(* Logix 5000 project; controller PBS_Perfusion vendor 1 type 14 code 217 rev 32.14; software revision 32.03; part 4 of 27 *)
(* tags used below, declared in another part *)
   ONS : DINT[3];
   REAL : DINT;

ADD_ON_INSTRUCTION AMP_Q_Segment_Execute   (* revision 1.0 *)
// Applied Motion - Q Segment Execute AOI
// Help:
// The SCL Command Execute AOI executes selected SCL commands (as listed under “Available SCL Commands” in the Host Command Reference).
VAR_IN_OUT
   Input : DINT[14]; {required}   // Drive Input Assembly
   Output : DINT[16]; {required}   // Drive Output Assembly
        [0]   // Command Word
        [1]   // Jog Speed (0.25 rev/min)
        [2]   // Jog Acceleration (10 rev/s/s)
        [3]   // Jog Deceleration (10 rev/s/s)
        [4]   // Point-to-Point Velocity (0.25 rev/min)
        [5]   // Point-to-Point Acceleration (10 rev/s/s)
        [6]   // Point-to-Point Deceleration (10 rev/s/s)
        [7]   // Point-to-Point Distance (Motor steps)
        [9]   // (2x ASCII Letters in 16 lower word)
        [10]   // Data/Register 1
        [11]   // Data/Register 2
END_VAR
VAR_INPUT
   RPI : DINT := 100; {visible}   // Drive Connection Request Packet Interval (milliseconds)
   LoadAndExec : BOOL; {required}   // Load and Execute the specified Q segment (edge triggered)
   Q_Segment : DINT; {required}   // Q Segment to Load and Execute
END_VAR
VAR_OUTPUT
   Sent : BOOL; {access Read Only, visible}   // Command has been sent to drive
   In_Progress : BOOL; {access Read Only, visible}   // In progress = sending command
   Done : BOOL; {access Read Only, visible}   // Command sent
   Error : BOOL; {access Read Only, visible}   // Command failed to be sent
   State : DINT := 10; {access Read Only}   // Internal state of progress
END_VAR
VAR
   Loc_StatusCode : AMP_Status_Word;
   Loc_CommandOff_Timer : TIMER;   // Timer to make sure command value was 0 before sending a new command
   Loc_CommandOn_Timer : TIMER;   // Timer to make sure command value is set long enough to be sent to drive
   Loc_Input_Assembly : AMP_Input_Assembly_v2; {access None}
   Loc_Start_ONS : BOOL; {access None}
END_VAR

ROUTINE Logic   (* ladder *)
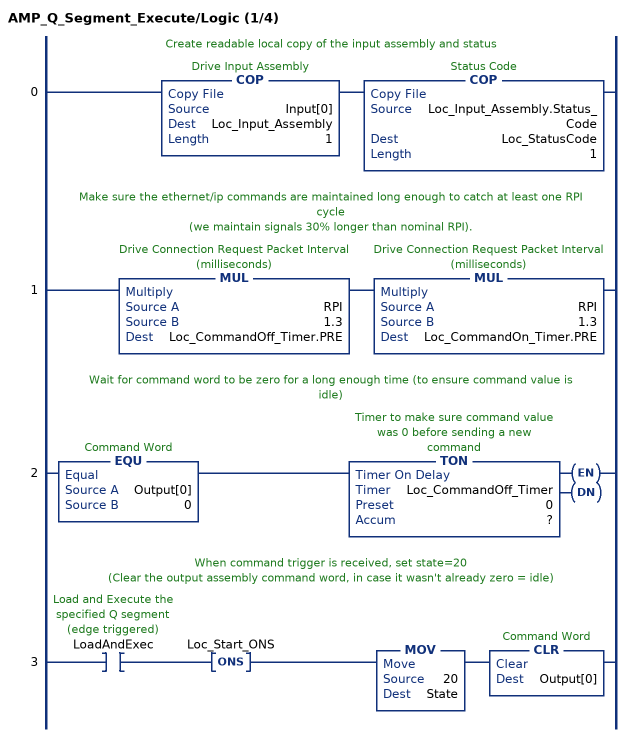
   // Create readable local copy of the input assembly and status
   0: COP(Input[0],Loc_Input_Assembly,1)COP(Loc_Input_Assembly.Status_Code,Loc_StatusCode,1);
   // Make sure the ethernet/ip commands are maintained long enough to catch at least one RPI cycle
   // (we maintain signals 30% longer than nominal RPI).
   1: MUL(RPI,1.3,Loc_CommandOff_Timer.PRE)MUL(RPI,1.3,Loc_CommandOn_Timer.PRE);
   // Wait for command word to be zero for a long enough time (to ensure command value is idle)
   2: EQU(Output[0],0)TON(Loc_CommandOff_Timer,?,?);
   // When command trigger is received, set state=20
   // (Clear the output assembly command word, in case it wasn't already zero = idle)
   3: XIC(LoadAndExec)ONS(Loc_Start_ONS)MOV(20,State)CLR(Output[0]);
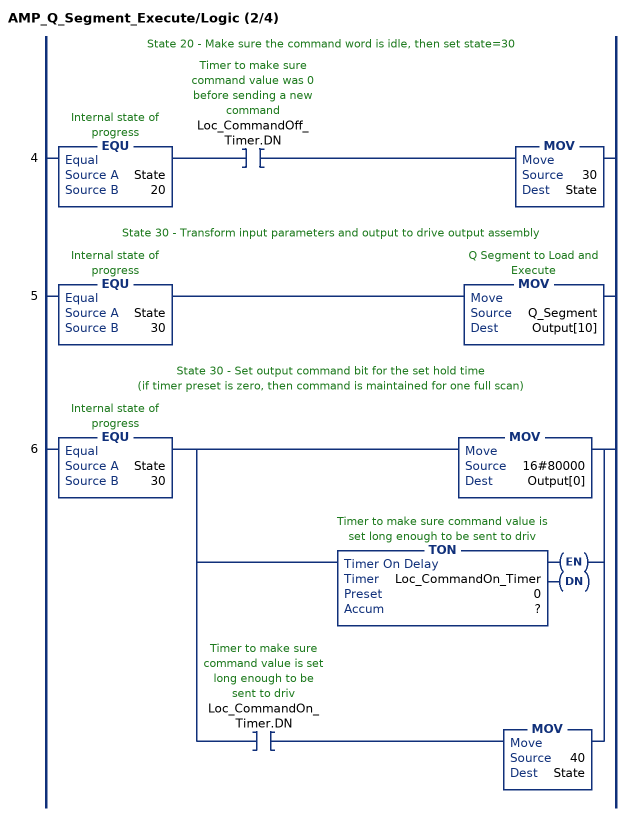
   // State 20 - Make sure the command word is idle, then set state=30
   4: EQU(State,20)XIC(Loc_CommandOff_Timer.DN)MOV(30,State);
   // State 30 - Transform input parameters and output to drive output assembly
   5: EQU(State,30)MOV(Q_Segment,Output[10]);
   // State 30 - Set output command bit for the set hold time
   // (if timer preset is zero, then command is maintained for one full scan)
   6: EQU(State,30)[MOV(16#80000,Output[0]) ,TON(Loc_CommandOn_Timer,?,?) ,XIC(Loc_CommandOn_Timer.DN) MOV(40,State) ];
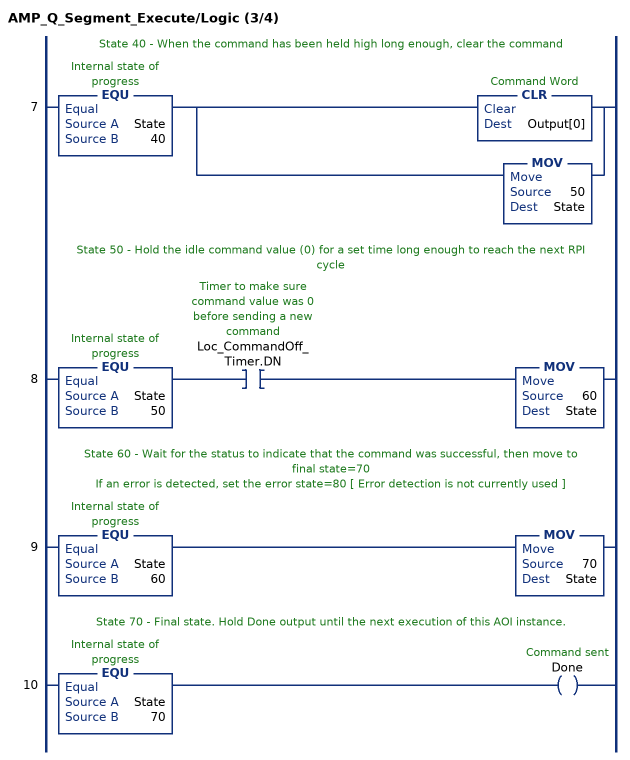
   // State 40 - When the command has been held high long enough, clear the command
   7: EQU(State,40)[CLR(Output[0]) ,MOV(50,State) ];
   // State 50 - Hold the idle command value (0) for a set time long enough to reach the next RPI cycle
   8: EQU(State,50)XIC(Loc_CommandOff_Timer.DN)MOV(60,State);
   // State 60 - Wait for the status to indicate that the command was successful, then move to final state=70
   // If an error is detected, set the error state=80 [ Error detection is not currently used ]
   9: EQU(State,60)MOV(70,State);
   // State 70 - Final state. Hold Done output until the next execution of this AOI instance.
   10: EQU(State,70)OTE(Done);
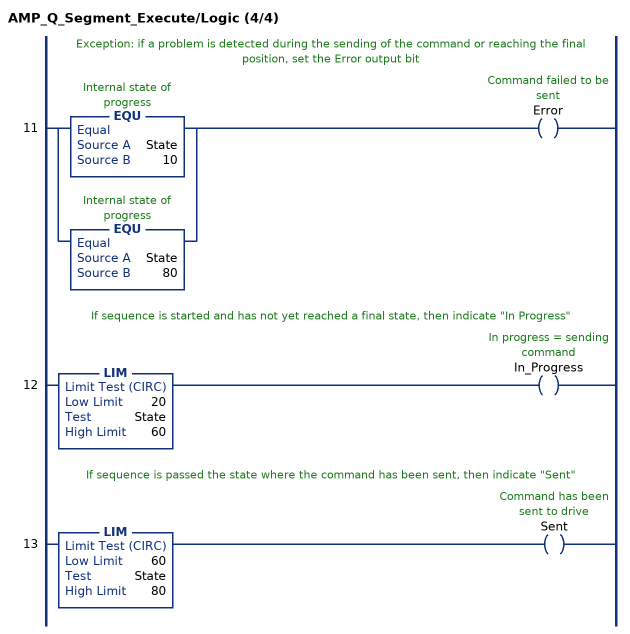
   // Exception: if a problem is detected during the sending of the command or reaching the final position, set the Error output bit
   11: [EQU(State,10) ,EQU(State,80) ]OTE(Error);
   // If sequence is started and has not yet reached a final state, then indicate "In Progress"
   12: LIM(20,State,60)OTE(In_Progress);
   // If sequence is passed the state where the command has been sent, then indicate "Sent"
   13: LIM(60,State,80)OTE(Sent);
END_ROUTINE
END_ADD_ON_INSTRUCTION

ADD_ON_INSTRUCTION AMP_Relative_Move   (* revision 1.0 *)
// Applied Motion - Relative Move AOI
// Help:
// The Relative Move AOI is used to move an axis by a specified distance (positive or negative) relative to its currently commanded position.
VAR_IN_OUT
   Input : DINT[14]; {required}   // Drive Input Assembly
   Output : DINT[16]; {required}   // Drive Output Assembly
        [0]   // Command Word
        [1]   // Jog Speed (0.25 rev/min)
        [2]   // Jog Acceleration (10 rev/s/s)
        [3]   // Jog Deceleration (10 rev/s/s)
        [4]   // Point-to-Point Velocity (0.25 rev/min)
        [5]   // Point-to-Point Acceleration (10 rev/min/s)
        [6]   // Point-to-Point Deceleration (10 rev/min/s)
        [7]   // Point-to-Point Distance (Motor steps)
        [9]   // (2x ASCII Letters in 16 lower word)
        [10]   // Data/Register 1
        [11]   // Data/Register 2
END_VAR
VAR_INPUT
   RPI : DINT := 100; {visible}   // Drive Connection Request Packet Interval (milliseconds)
   Start : BOOL; {required}   // Start the Relative Move
   Distance : DINT; {required}   // Relative Distance to Move (steps, negative = reverse)
   Speed : REAL; {required}   // Velocity of Move (rev/min)
   Acc : REAL; {required}   // Acceleration of Move (rev/s/s)
   Dec : REAL; {required}   // Deceleration (rev/s/s)
END_VAR
VAR_OUTPUT
   Sent : BOOL; {access Read Only, visible}   // Move has been sent to drive
   In_Progress : BOOL; {access Read Only, visible}   // Move in progress
   Done : BOOL; {access Read Only, visible}   // Move completed without errors - desired position reached
   Error : BOOL; {access Read Only, visible}   // Move failed to complete - drive not ready or faulted
   State : DINT := 10; {access Read Only}   // Internal state of progress
END_VAR
VAR
   Loc_StatusCode : AMP_Status_Word;
   Loc_CommandOff_Timer : TIMER;   // Timer to make sure command value was 0 before sending a new command
   Loc_CommandOn_Timer : TIMER;   // Timer to make sure command value is set long enough to be sent to drive
   Loc_Input_Assembly : AMP_Input_Assembly_v2; {access None}
   Loc_Start_ONS : BOOL; {access None}
   Loc_AlarmCode : AMP_Alarm_Word; {access None}
END_VAR

ROUTINE Logic   (* ladder *)
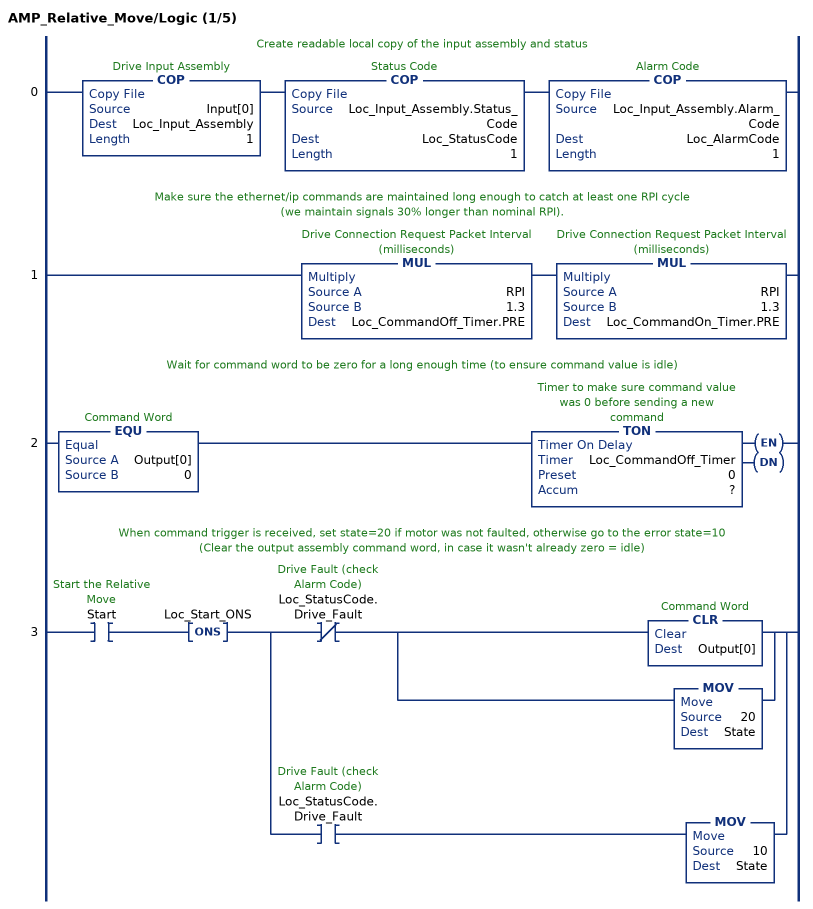
   // Create readable local copy of the input assembly and status
   0: COP(Input[0],Loc_Input_Assembly,1)COP(Loc_Input_Assembly.Status_Code,Loc_StatusCode,1)COP(Loc_Input_Assembly.Alarm_Code,Loc_AlarmCode,1);
   // Make sure the ethernet/ip commands are maintained long enough to catch at least one RPI cycle
   // (we maintain signals 30% longer than nominal RPI).
   1: MUL(RPI,1.3,Loc_CommandOff_Timer.PRE)MUL(RPI,1.3,Loc_CommandOn_Timer.PRE);
   // Wait for command word to be zero for a long enough time (to ensure command value is idle)
   2: EQU(Output[0],0)TON(Loc_CommandOff_Timer,?,?);
   // When command trigger is received, set state=20 if motor was not faulted, otherwise go to the error state=10
   // (Clear the output assembly command word, in case it wasn't already zero = idle)
   3: XIC(Start)ONS(Loc_Start_ONS)[XIO(Loc_StatusCode.Drive_Fault) [CLR(Output[0]) ,MOV(20,State) ] ,XIC(Loc_StatusCode.Drive_Fault) MOV(10,State) ];
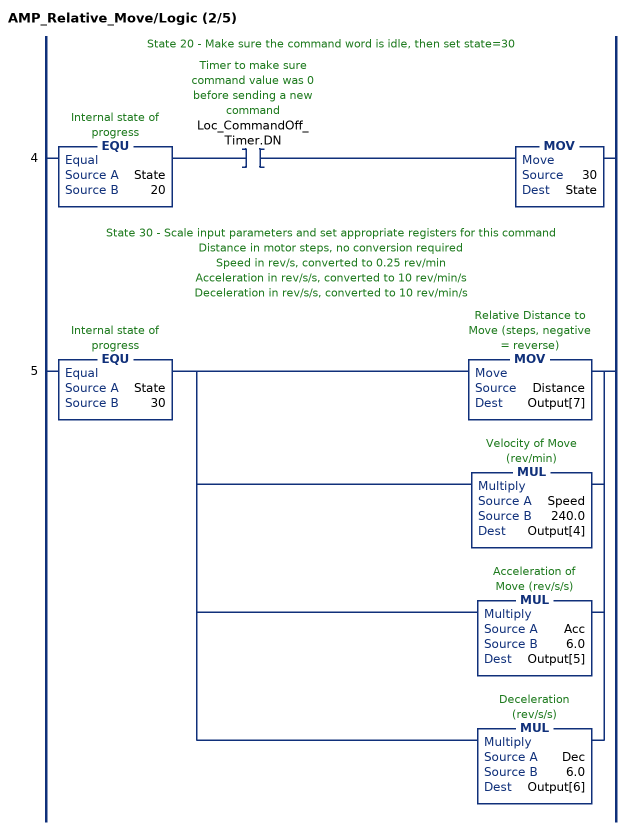
   // State 20 - Make sure the command word is idle, then set state=30
   4: EQU(State,20)XIC(Loc_CommandOff_Timer.DN)MOV(30,State);
   // State 30 - Scale input parameters and set appropriate registers for this command
   // Distance in motor steps, no conversion required
   // Speed in rev/s, converted to 0.25 rev/min
   // Acceleration in rev/s/s, converted to 10 rev/min/s
   // Deceleration in rev/s/s, converted to 10 rev/min/s
   5: EQU(State,30)[MOV(Distance,Output[7]) ,MUL(Speed,240.0,Output[4]) ,MUL(Acc,6.0,Output[5]) ,MUL(Dec,6.0,Output[6]) ];
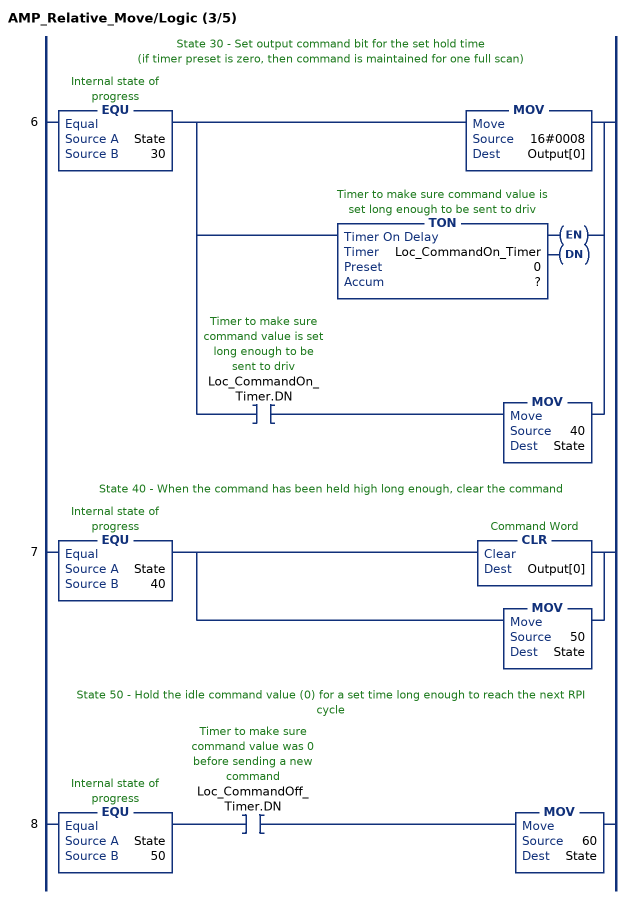
   // State 30 - Set output command bit for the set hold time
   // (if timer preset is zero, then command is maintained for one full scan)
   6: EQU(State,30)[MOV(16#0008,Output[0]) ,TON(Loc_CommandOn_Timer,?,?) ,XIC(Loc_CommandOn_Timer.DN) MOV(40,State) ];
   // State 40 - When the command has been held high long enough, clear the command
   7: EQU(State,40)[CLR(Output[0]) ,MOV(50,State) ];
   // State 50 - Hold the idle command value (0) for a set time long enough to reach the next RPI cycle
   8: EQU(State,50)XIC(Loc_CommandOff_Timer.DN)MOV(60,State);
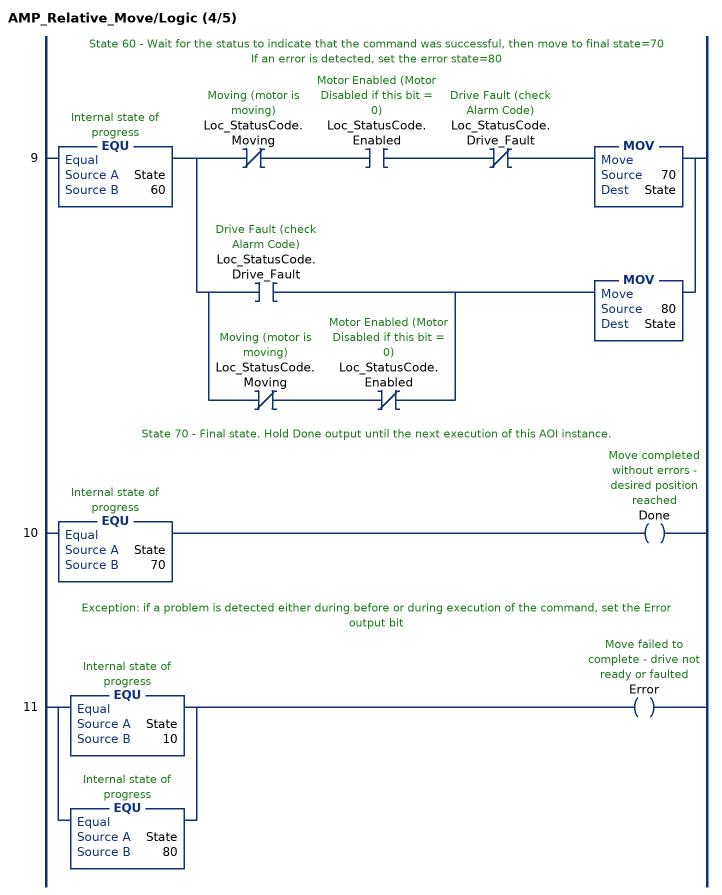
   // State 60 - Wait for the status to indicate that the command was successful, then move to final state=70
   // If an error is detected, set the error state=80
   9: EQU(State,60)[XIO(Loc_StatusCode.Moving) XIC(Loc_StatusCode.Enabled) XIO(Loc_StatusCode.Drive_Fault) MOV(70,State) ,[XIC(Loc_StatusCode.Drive_Fault) ,XIO(Loc_StatusCode.Moving) XIO(Loc_StatusCode.Enabled) ] MOV(80,State) ];
   // State 70 - Final state. Hold Done output until the next execution of this AOI instance.
   10: EQU(State,70)OTE(Done);
   // Exception: if a problem is detected either during before or during execution of the command, set the Error output bit
   11: [EQU(State,10) ,EQU(State,80) ]OTE(Error);
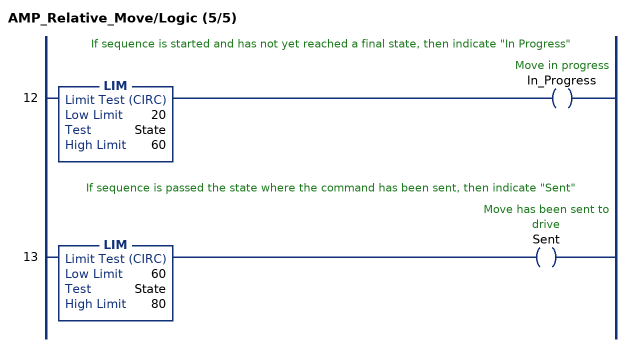
   // If sequence is started and has not yet reached a final state, then indicate "In Progress"
   12: LIM(20,State,60)OTE(In_Progress);
   // If sequence is passed the state where the command has been sent, then indicate "Sent"
   13: LIM(60,State,80)OTE(Sent);
END_ROUTINE
END_ADD_ON_INSTRUCTION

ADD_ON_INSTRUCTION AMP_Status_Code   (* revision 1.0 *)
// Applied Motion - Status Code AOI
// Help:
// The Status Code AOI uses the raw data stored in the Status Code word (Element 0 from Input Assembly 0x65) to set individual appropriately named boolean outputs.
VAR_INPUT
   Input : DINT; {required}   // Element 0 from Drive Input Assembly (0x65)
END_VAR
VAR_OUTPUT
   Motor_Enabled : BOOL; {access Read Only, visible}
   Sampling : BOOL; {access Read Only, visible}
   Drive_Fault : BOOL; {access Read Only, visible}
   In_Position : BOOL; {access Read Only, visible}
   Moving : BOOL; {access Read Only, visible}
   Jogging : BOOL; {access Read Only, visible}
   Stopping : BOOL; {access Read Only, visible}
   Waiting : BOOL; {access Read Only, visible}
   Saving : BOOL; {access Read Only, visible}
   Alarm_Present : BOOL; {access Read Only, visible}
   Homing : BOOL; {access Read Only, visible}
   Wait_Time : BOOL; {access Read Only, visible}
   Wizard_Running : BOOL; {access Read Only, visible}
   Checking_Encoder : BOOL; {access Read Only, visible}
   Q_Program_Running : BOOL; {access Read Only, visible}
   Initializing : BOOL; {access Read Only, visible}
END_VAR

ROUTINE Logic   (* ladder *)
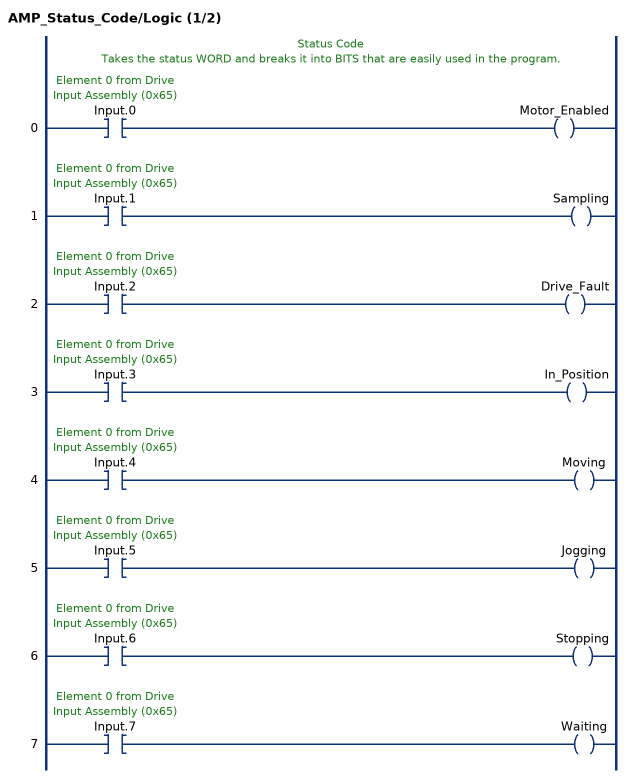
   // Status Code
   // Takes the status WORD and breaks it into BITS that are easily used in the program.
   0: XIC(Input.0)OTE(Motor_Enabled);
   1: XIC(Input.1)OTE(Sampling);
   2: XIC(Input.2)OTE(Drive_Fault);
   3: XIC(Input.3)OTE(In_Position);
   4: XIC(Input.4)OTE(Moving);
   5: XIC(Input.5)OTE(Jogging);
   6: XIC(Input.6)OTE(Stopping);
   7: XIC(Input.7)OTE(Waiting);
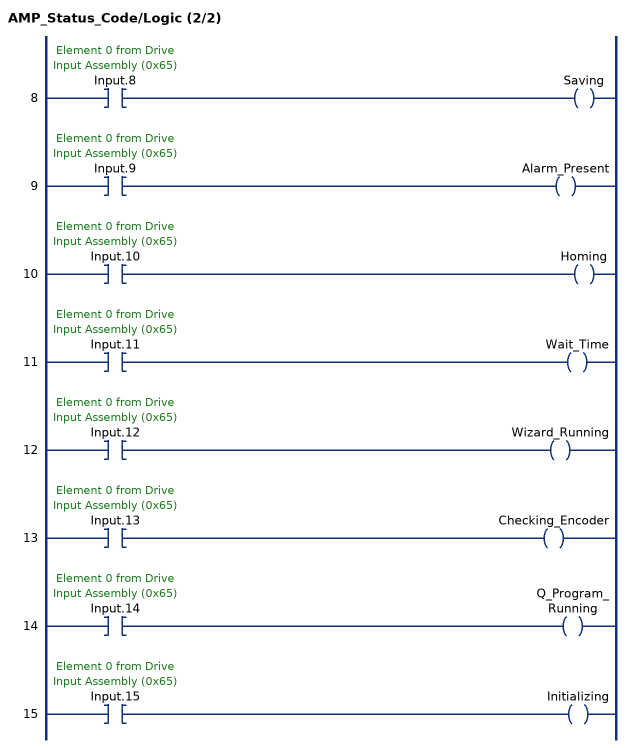
   8: XIC(Input.8)OTE(Saving);
   9: XIC(Input.9)OTE(Alarm_Present);
   10: XIC(Input.10)OTE(Homing);
   11: XIC(Input.11)OTE(Wait_Time);
   12: XIC(Input.12)OTE(Wizard_Running);
   13: XIC(Input.13)OTE(Checking_Encoder);
   14: XIC(Input.14)OTE(Q_Program_Running);
   15: XIC(Input.15)OTE(Initializing);
END_ROUTINE
END_ADD_ON_INSTRUCTION

ADD_ON_INSTRUCTION AMP_Tuning_Params_StepSERVO   (* revision 1.0 *)
// Applied Motion - Tuning Parameters StepSERVO AOI
// Help:
// The Tuning Parameters for StepSERVO AOI accepts all the required parameters for SCL commands VP, VI, KK, KC, KP, KD and KE, and then scales and issues these to the drive, one at a time.
VAR_IN_OUT
   MSG_Write : SINT[8]; {required}   // Message Write data tag
        [0]   // Message Reserved = 0
        [1]   // Message Type (16#01 or 16#02)
        [2]   // Type 1: Register Type 2: Opcode
        [3]   // Type 1: Opcode Type 2: Operand
        [4]   // Type 1: Parameter 1 Type 2: data MSB
        [5]   // Type 1: Parameter 2 Type 2: data LSB
        [6]   // Type 1: Parameter 3 Type 2: not used
        [7]   // Type 1: Parameter 4 Type 2: not used
   SendMsg : MESSAGE; {required}   // Message tag
   MSG_Response : SINT[8]; {required}   // Message Response data tag
        [0]   // Command Word
        [1]   // Jog Speed (0.25 rev/min)
        [2]   // Jog Acceleration (10 rev/s/s)
        [3]   // Jog Deceleration (10 rev/s/s)
        [4]   // Point-to-Point Velocity (0.25 rev/min)
        [5]   // Point-to-Point Acceleration (10 rev/s/s)
        [6]   // Point-to-Point Deceleration (10 rev/s/s)
        [7]   // Point-to-Point Distance (Motor steps)
END_VAR
VAR_INPUT
   Configure : BOOL; {required}   // Start the Configuration
   VP : INT; {required}   // Velocity Mode Proportional Constant
   VI : INT; {required}   // Velocity Integrator Constant
   KP : INT; {required}   // Proportional Global Gain Value
   KK : INT; {required}   // Inertia Feedforward Gain
   KE : INT; {required}   // Differential Filter Gain Value
   KD : INT; {required}   // Damping Gain Value
   KC : INT; {required}   // Overall Servo Filter value
END_VAR
VAR_OUTPUT
   Sent : BOOL; {access Read Only, visible}   // All parameter settings have been sent to drive
   In_Progress : BOOL; {access Read Only, visible}   // The setting of parameters is in progress
   Done : BOOL; {access Read Only, visible}   // Parameters set without errors
   Error : BOOL; {access Read Only, visible}   // Configuration failed to complete - drive not ready or faulted
   State : DINT := 34; {access Read Only}   // Internal state of progress
END_VAR
VAR
   Loc_Start_ONS : BOOL; {access None}
   MSG_Active : BOOL;
END_VAR

ROUTINE Logic   (* ladder *)
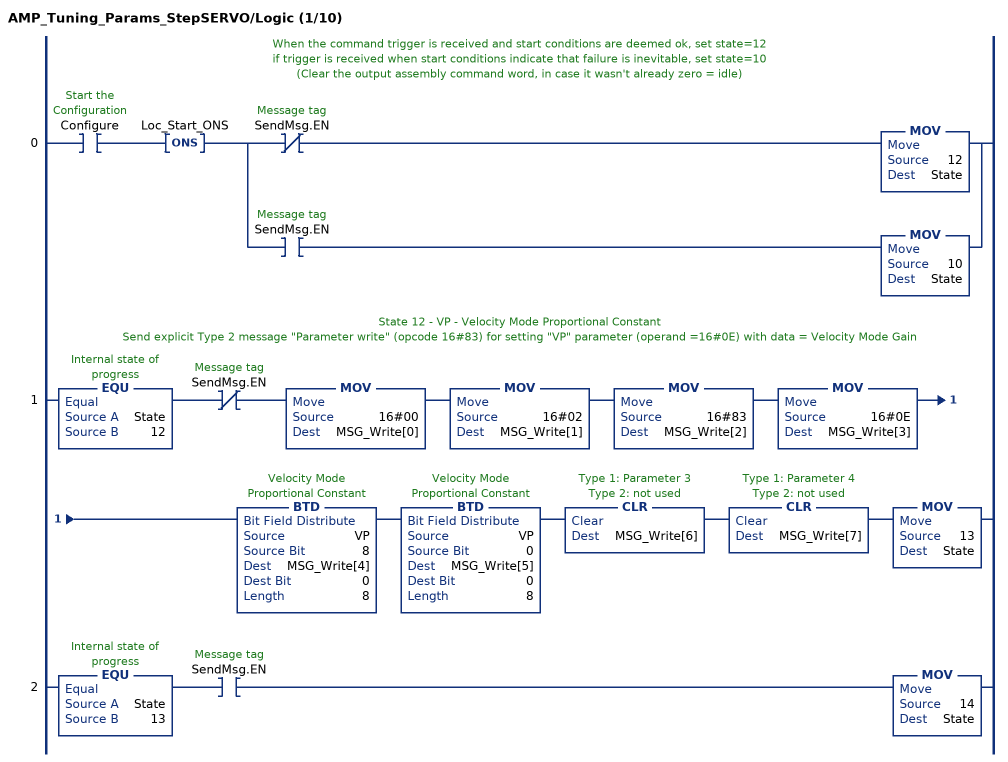
   // When the command trigger is received and start conditions are deemed ok, set state=12
   // if trigger is received when start conditions indicate that failure is inevitable, set state=10
   // (Clear the output assembly command word, in case it wasn't already zero = idle)
   0: XIC(Configure)ONS(Loc_Start_ONS)[XIO(SendMsg.EN) MOV(12,State) ,XIC(SendMsg.EN) MOV(10,State) ];
   // State 12 - VP - Velocity Mode Proportional Constant
   // Send explicit Type 2 message "Parameter write" (opcode 16#83) for setting "VP" parameter (operand =16#0E) with data = Velocity Mode Gain
   1: EQU(State,12)XIO(SendMsg.EN)MOV(16#00,MSG_Write[0])MOV(16#02,MSG_Write[1])MOV(16#83,MSG_Write[2])MOV(16#0E,MSG_Write[3])BTD(VP,8,MSG_Write[4],0,8)BTD(VP,0,MSG_Write[5],0,8)CLR(MSG_Write[6])CLR(MSG_Write[7])MOV(13,State);
   2: EQU(State,13)XIC(SendMsg.EN)MOV(14,State);
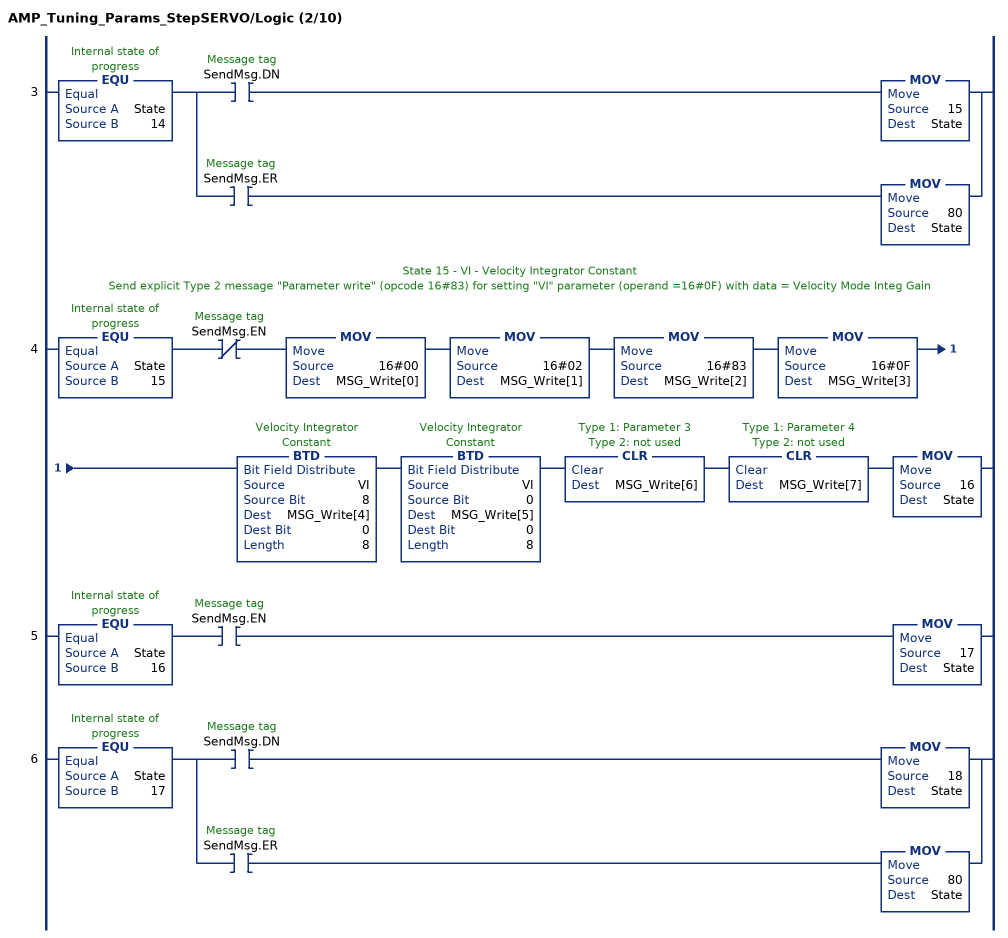
   3: EQU(State,14)[XIC(SendMsg.DN) MOV(15,State) ,XIC(SendMsg.ER) MOV(80,State) ];
   // State 15 - VI - Velocity Integrator Constant
   // Send explicit Type 2 message "Parameter write" (opcode 16#83) for setting "VI" parameter (operand =16#0F) with data = Velocity Mode Integ Gain
   4: EQU(State,15)XIO(SendMsg.EN)MOV(16#00,MSG_Write[0])MOV(16#02,MSG_Write[1])MOV(16#83,MSG_Write[2])MOV(16#0F,MSG_Write[3])BTD(VI,8,MSG_Write[4],0,8)BTD(VI,0,MSG_Write[5],0,8)CLR(MSG_Write[6])CLR(MSG_Write[7])MOV(16,State);
   5: EQU(State,16)XIC(SendMsg.EN)MOV(17,State);
   6: EQU(State,17)[XIC(SendMsg.DN) MOV(18,State) ,XIC(SendMsg.ER) MOV(80,State) ];
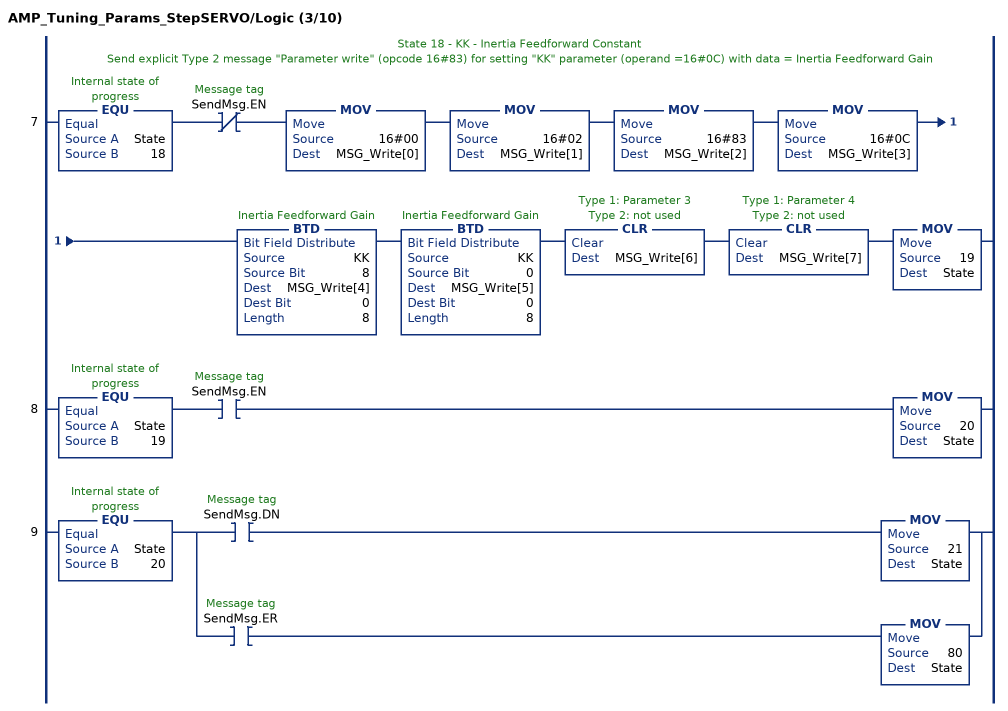
   // State 18 - KK - Inertia Feedforward Constant
   // Send explicit Type 2 message "Parameter write" (opcode 16#83) for setting "KK" parameter (operand =16#0C) with data = Inertia Feedforward Gain
   7: EQU(State,18)XIO(SendMsg.EN)MOV(16#00,MSG_Write[0])MOV(16#02,MSG_Write[1])MOV(16#83,MSG_Write[2])MOV(16#0C,MSG_Write[3])BTD(KK,8,MSG_Write[4],0,8)BTD(KK,0,MSG_Write[5],0,8)CLR(MSG_Write[6])CLR(MSG_Write[7])MOV(19,State);
   8: EQU(State,19)XIC(SendMsg.EN)MOV(20,State);
   9: EQU(State,20)[XIC(SendMsg.DN) MOV(21,State) ,XIC(SendMsg.ER) MOV(80,State) ];
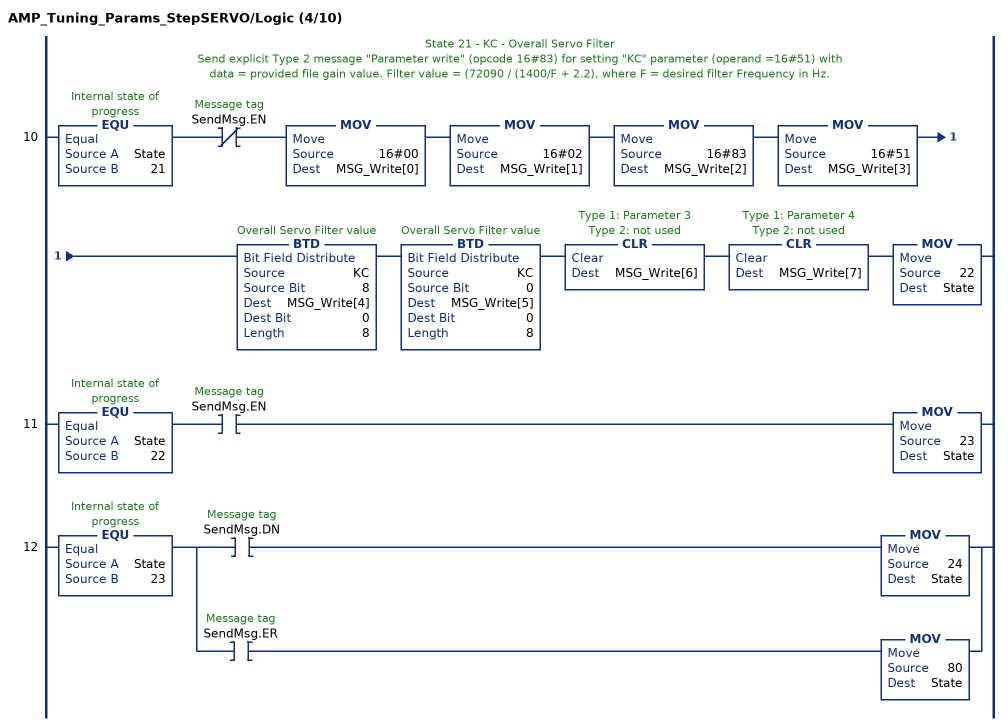
   // State 21 - KC - Overall Servo Filter
   // Send explicit Type 2 message "Parameter write" (opcode 16#83) for setting "KC" parameter (operand =16#51) with
   // data = provided file gain value. Filter value = (72090 / (1400/F + 2.2), where F = desired filter Frequency in Hz.
   10: EQU(State,21)XIO(SendMsg.EN)MOV(16#00,MSG_Write[0])MOV(16#02,MSG_Write[1])MOV(16#83,MSG_Write[2])MOV(16#51,MSG_Write[3])BTD(KC,8,MSG_Write[4],0,8)BTD(KC,0,MSG_Write[5],0,8)CLR(MSG_Write[6])CLR(MSG_Write[7])MOV(22,State);
   11: EQU(State,22)XIC(SendMsg.EN)MOV(23,State);
   12: EQU(State,23)[XIC(SendMsg.DN) MOV(24,State) ,XIC(SendMsg.ER) MOV(80,State) ];
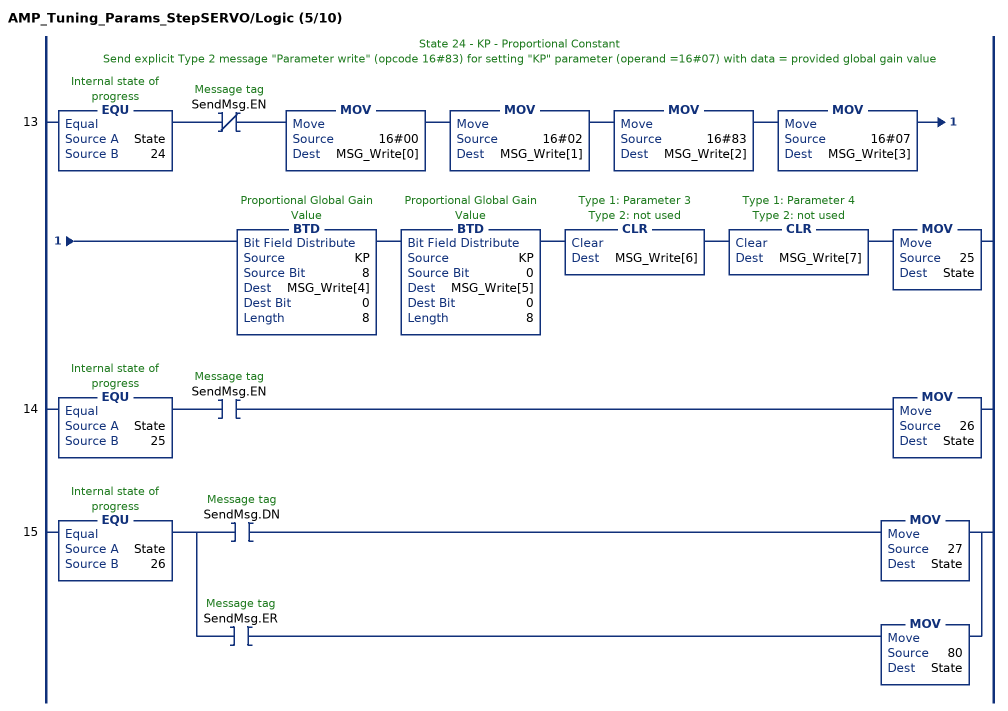
   // State 24 - KP - Proportional Constant
   // Send explicit Type 2 message "Parameter write" (opcode 16#83) for setting "KP" parameter (operand =16#07) with data = provided global gain value
   13: EQU(State,24)XIO(SendMsg.EN)MOV(16#00,MSG_Write[0])MOV(16#02,MSG_Write[1])MOV(16#83,MSG_Write[2])MOV(16#07,MSG_Write[3])BTD(KP,8,MSG_Write[4],0,8)BTD(KP,0,MSG_Write[5],0,8)CLR(MSG_Write[6])CLR(MSG_Write[7])MOV(25,State);
   14: EQU(State,25)XIC(SendMsg.EN)MOV(26,State);
   15: EQU(State,26)[XIC(SendMsg.DN) MOV(27,State) ,XIC(SendMsg.ER) MOV(80,State) ];
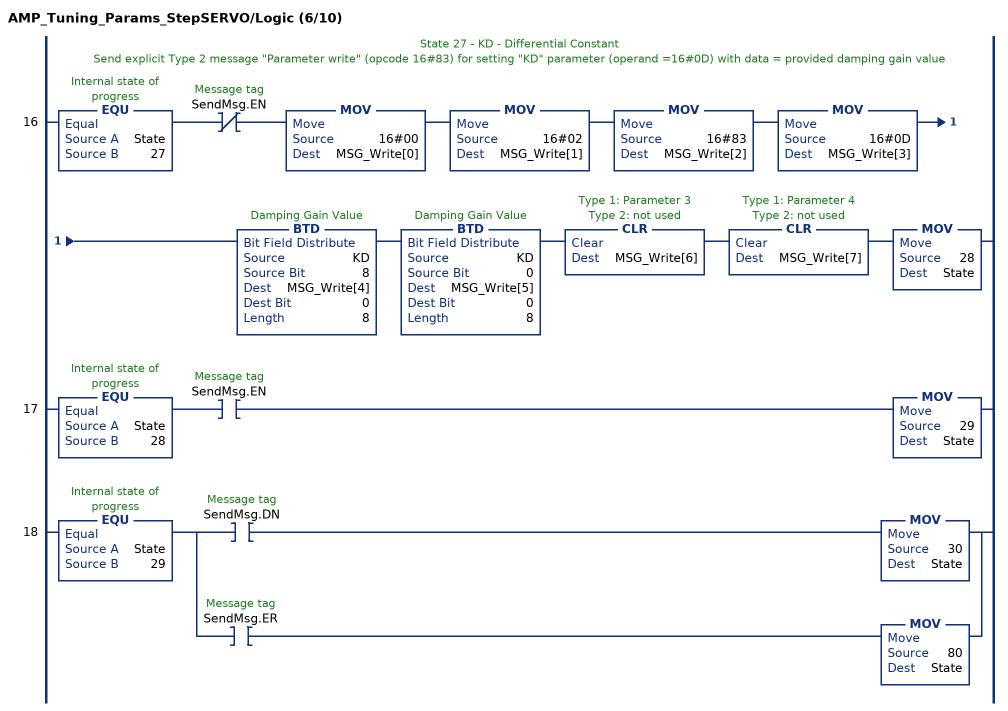
   // State 27 - KD - Differential Constant
   // Send explicit Type 2 message "Parameter write" (opcode 16#83) for setting "KD" parameter (operand =16#0D) with data = provided damping gain value
   16: EQU(State,27)XIO(SendMsg.EN)MOV(16#00,MSG_Write[0])MOV(16#02,MSG_Write[1])MOV(16#83,MSG_Write[2])MOV(16#0D,MSG_Write[3])BTD(KD,8,MSG_Write[4],0,8)BTD(KD,0,MSG_Write[5],0,8)CLR(MSG_Write[6])CLR(MSG_Write[7])MOV(28,State);
   17: EQU(State,28)XIC(SendMsg.EN)MOV(29,State);
   18: EQU(State,29)[XIC(SendMsg.DN) MOV(30,State) ,XIC(SendMsg.ER) MOV(80,State) ];
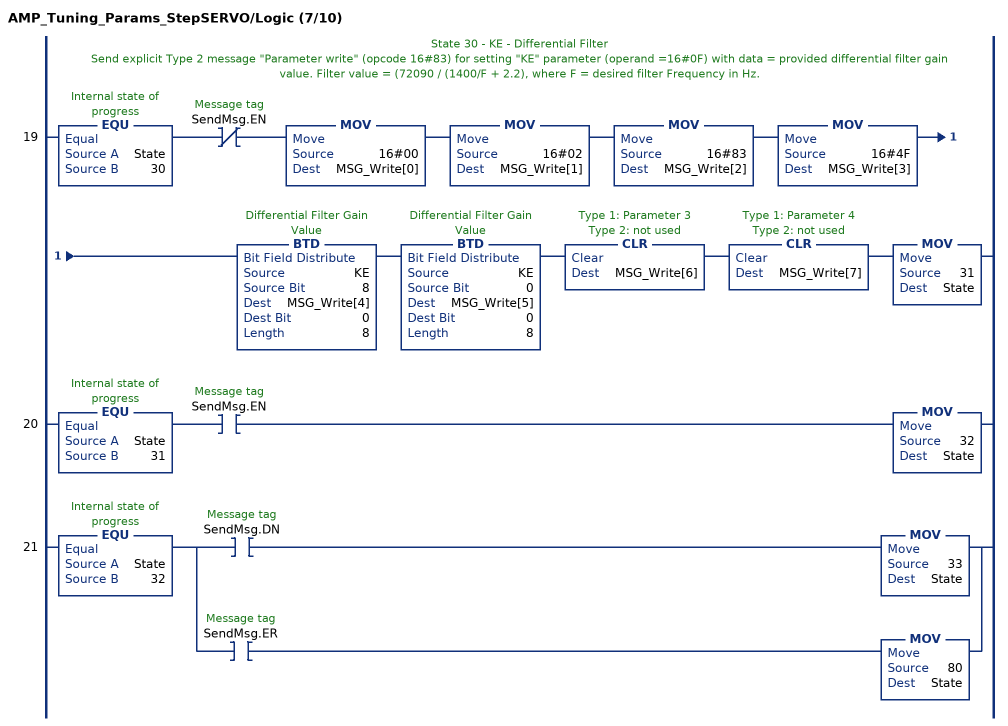
   // State 30 - KE - Differential Filter
   // Send explicit Type 2 message "Parameter write" (opcode 16#83) for setting "KE" parameter (operand =16#0F) with data = provided differential filter gain value. Filter value = (72090 / (1400/F + 2.2), where F = desired filter Frequency in Hz.
   19: EQU(State,30)XIO(SendMsg.EN)MOV(16#00,MSG_Write[0])MOV(16#02,MSG_Write[1])MOV(16#83,MSG_Write[2])MOV(16#4F,MSG_Write[3])BTD(KE,8,MSG_Write[4],0,8)BTD(KE,0,MSG_Write[5],0,8)CLR(MSG_Write[6])CLR(MSG_Write[7])MOV(31,State);
   20: EQU(State,31)XIC(SendMsg.EN)MOV(32,State);
   21: EQU(State,32)[XIC(SendMsg.DN) MOV(33,State) ,XIC(SendMsg.ER) MOV(80,State) ];
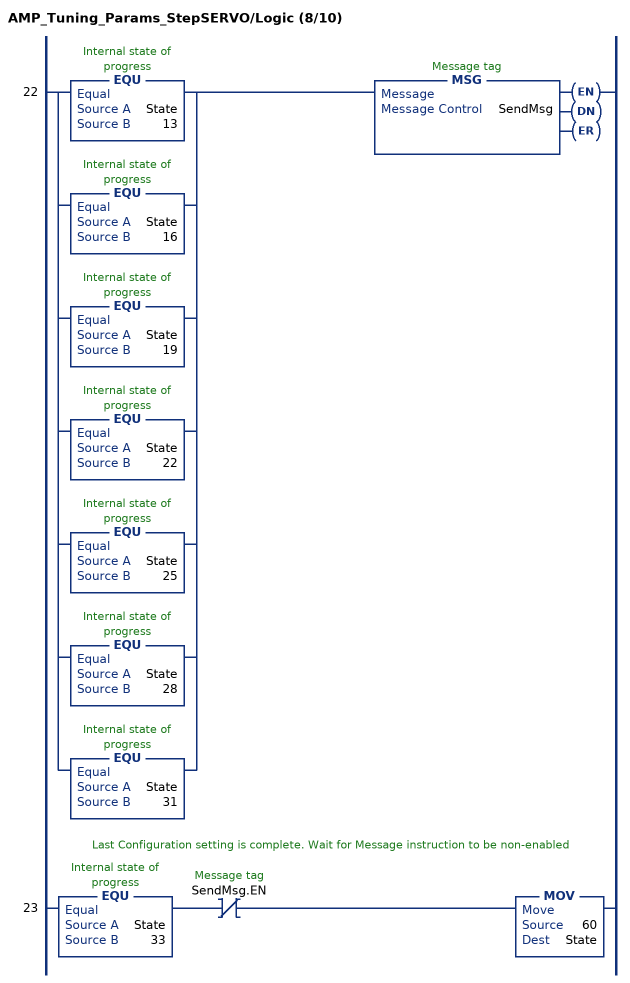
   22: [EQU(State,13) ,EQU(State,16) ,EQU(State,19) ,EQU(State,22) ,EQU(State,25) ,EQU(State,28) ,EQU(State,31) ]MSG(SendMsg);
   // Last Configuration setting is complete. Wait for Message instruction to be non-enabled
   23: EQU(State,33)XIO(SendMsg.EN)MOV(60,State);
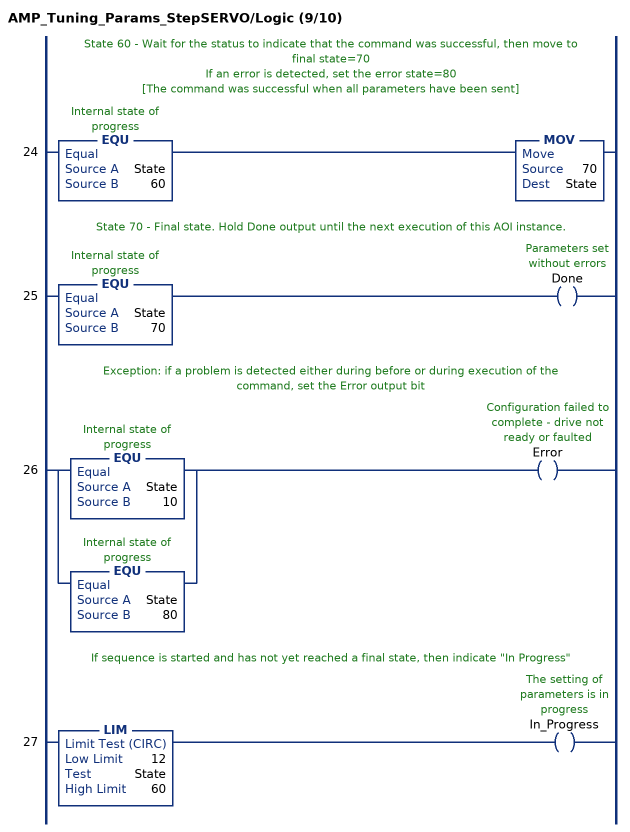
   // State 60 - Wait for the status to indicate that the command was successful, then move to final state=70
   // If an error is detected, set the error state=80
   // [The command was successful when all parameters have been sent]
   24: EQU(State,60)MOV(70,State);
   // State 70 - Final state. Hold Done output until the next execution of this AOI instance.
   25: EQU(State,70)OTE(Done);
   // Exception: if a problem is detected either during before or during execution of the command, set the Error output bit
   26: [EQU(State,10) ,EQU(State,80) ]OTE(Error);
   // If sequence is started and has not yet reached a final state, then indicate "In Progress"
   27: LIM(12,State,60)OTE(In_Progress);
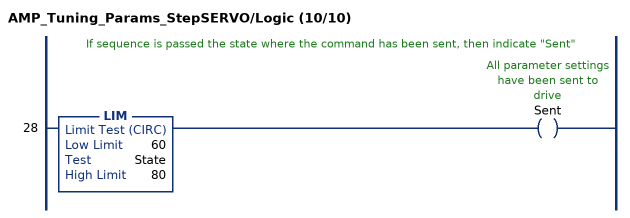
   // If sequence is passed the state where the command has been sent, then indicate "Sent"
   28: LIM(60,State,80)OTE(Sent);
END_ROUTINE
END_ADD_ON_INSTRUCTION
